INTERFACE I_Pizza

METHOD GetDescription : STRING
VAR_INPUT
END_VAR
END_METHOD

METHOD GetPrice : LREAL
VAR_INPUT
END_VAR
END_METHOD

END_INTERFACE

(* stored: Version 1.1.0.1, ProductVersion 3.1.4022.16
   Itf I_Pizza: Id {75d38bd0-716f-490c-807a-4daa8f26e0d3}
   Method GetDescription: Id {dd561ff2-195f-4c97-a177-50684d9b836f}
   Method GetPrice: Id {edeb25c6-511a-430c-a4d9-e87e27c3eec1} *)
